FUNCTION_BLOCK Test_WriteBySymbolName EXTENDS TUnitTestBase
VAR
    AdsWriteBySymbolName : TAdsWriteBySymbolName;
    ValueToWrite : INT := 3456;
    WriteResult : INT;
    ScanCount : DINT;
    State: INT;
END_VAR

CASE State OF
    0:
        ValueToWrite := 3456;
        WriteResult := 0;
        ScanCount := 0;
    
        AdsWriteBySymbolName.Execute(
            AmsNetId:= '', 
            Port:= 851, 
            SymbolName:= 'PB_TestRunner.Test_WriteBySymbolName.WriteResult', 
            WriteDataAddress:= ADR(ValueToWrite), 
            WriteDataLength:= SIZEOF(ValueToWrite), 
            KeepSymbolHandle:= FALSE);

        State := 10;
        
    10:
        ScanCount := ScanCount + 1;
        IF NOT AdsWriteBySymbolName.Execution.Busy THEN
            State := 20;    
		END_IF
        
    20:
        Assertion.AssertEquals_INT(
            Expected     := 3456,
            Actual       := WriteResult,
            ObjectName   := _TestName,
            Variablename := 'WriteResult'); 
 
        TestFinished();
        State := 0;
END_CASE

AdsWriteBySymbolName();

END_FUNCTION_BLOCK

(* stored: Version 1.1.0.1, ProductVersion 3.1.4024.3
   POU Test_WriteBySymbolName: Id {5311daf6-9f8e-00c7-03d0-f7ac73ec095f}, SpecialFunc None *)
